Yaskawa INFORM job: 3-ZMP.JBI

/JOB
//NAME 3-ZMP
///FOLDERNAME INNE
//POS
///NPOS 2,2,0,0,0,0
///TOOL 0
///POSTYPE PULSE
///PULSE
C00000=-1207,-5179,111529,-786,38079,299
C00001=-2344,-185080,-108491,-822,81027,-287
BC00000=277960,1059793,995145
BC00001=277960,1059793,324739
//INST
///DATE 2023/10/04 15:13
///ATTR SC,RW
///GROUP1 RB1,BS1
NOP
MOVJ C00000 BC00000 VJ=0.78
MOVJ C00001 BC00001 VJ=0.78
END
